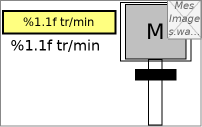
VISUALIZATION VISU_PS  // 202x127
VAR_IN_OUT
	m_Input_MOTOR : BLOCK_VARIATEUR_MOTEUR;
END_VAR
    Rectangle (148,59 14x66)
    RoundedRectangle (125,4 61x55), "M", colour toggle: (m_Input_MOTOR.STATE_On) <> 0
    Rectangle (3,34 112x23), "%1.1f tr/min", text variable: m_Input_MOTOR.STATE_Consigne, invisible if: TRUE
    RoundedRectangle (2,10 114x24), "%1.1f tr/min", text variable: m_Input_MOTOR.PRM_Cons_Vitesse, input disabled if: NOT Global_Variables.PRG_USER.ACTU_USER.MAINTENANCE OR NOT m_Input_MOTOR.Manual
        OnMouseDown: write the text variable via InputWithLimits, min 0.2, max 20.0
    Rectangle (135,69 41x11)
    Rectangle (120,2 71x59), invisible if: NOT (m_Input_MOTOR.Autor_OFF_IHM) OR NOT PRG_User.ACTU_USER.MAINTENANCE
        tap m_Input_MOTOR.M_OFF
    Rectangle (120,2 71x59), invisible if: NOT (m_Input_MOTOR.Autor_ON_IHM) OR NOT PRG_User.ACTU_USER.MAINTENANCE
        tap m_Input_MOTOR.M_ON
    Image (167,-2 35x41), invisible if: NOT m_Input_MOTOR.STATE_NOK, image: MesImages.warning
END_VISUALIZATION

(* stored: Version 1.1.0.1, ProductVersion 3.1.4024.10
   Visu VISU_PS: Id {f7bdf436-2605-4576-a89c-f237bffcd5ed} *)
